// TIA Portal project "этикетка" (V15.1)

(* hardware
DEVICE "Станция S7-1200_1"  S7-1200 Station
   slot 0: "Rack_0"  S7-1200 Rack  Rack  V1.0
   slot 1: "PLC_1"  CPU 1215C DC/DC/DC  6ES7 215-1AG40-0XB0  V4.2
   slot 3: "DQ 4x5 В пост. тока_1"  DQ4 signal board (200 kHz)  6ES7 222-1AD30-0XB0  V1.0
*)

// ===== PLC "PLC_1"  CPU 1215C DC/DC/DC =====

VAR_GLOBAL   // PLC tag table "Стандартная таблица переменных"
   ""ручной режим/наладка"" AT %I0.0 : Bool;
   ""старт"" AT %I0.3 : Bool;
   ""стоп"" AT %I0.4 : Bool;
   ""аварийный стоп"" AT %I0.7 : Bool;
   ""датчик этикетки"" AT %I0.2 : Bool;
   ""датчик ампулы"" AT %I0.1 : Bool;
   ""Tag_31"" AT %I1.5 : Bool;
   ""скорость транспортера"" AT %QW64 : Word;
   ""старт транспортера"" AT %Q0.0 : Bool;
   ""скорость прикатки"" AT %QW66 : Word;
   ""старт прикатки"" AT %Q0.1 : Bool;
   ""Tag_8"" AT %Q4.1 : Bool;
   ""Axis_1_Импульс"" AT %Q4.0 : Bool;
   ""Tag_26"" AT %Q0.3 : Bool;
   ""printer"" AT %Q0.2 : Bool;
END_VAR